INTERFACE I_Motor

END_INTERFACE

(* stored: Version 1.1.0.1, ProductVersion 3.1.4024.16
   Itf I_Motor: Id {926770be-804f-46bd-b05e-5e636180ea19} *)
